FUNCTION_BLOCK PressureBuildUp
VAR
	fbPressureGradient : PressureGradient;
	fbDiscreteIntegrator : DiscreteIntegrator;
	
	IntegratorIn : LREAL;
	IntegratorOut : LREAL;
	ssMethodType : SINT := 1; 
	

//	fbPressure : DiscreteIntegrator;
//	fbPressureGradient : PressureGradient;
END_VAR
VAR_INPUT
	TotalVolume1 : LREAL;
	FlowrateIn1 : LREAL;
	FlowrateOut1 : LREAL;
	par : ST_pValveControlledCylinder;
END_VAR
VAR_OUTPUT
//	PressureBar : LREAL;
//	PressurePascal : LREAL;
END_VAR


fbPressureGradient(
	TotalVolume := TotalVolume1,
	FlowrateIn := FlowrateIn1,
	FlowrateOut := FlowrateOut1
	);

//pA
(* fbPressure(
	ssMethodType := ssMethodType,
	In1 := fbPressureGradient.PressureGradientPascal,
	Out1 => PressurePascal
	);
	
PressureGradientPascal := PressureGradientBar*1E5;      //Multiplies to get Pascal *)

END_FUNCTION_BLOCK

(* stored: Version 1.1.0.1, ProductVersion 3.1.4024.9
   POU PressureBuildUp: Id {464e8b07-8a4d-4793-8528-94ac640820e4}, SpecialFunc None *)
